(* Name: Nhat Ha Pham
   Student number: 547508*)

FUNCTION_BLOCK fbMaking_Coffee
VAR_INPUT
	GetOffBed : BOOL;  
	HeatButton : BOOL;
	Start : BOOL;
	ToastState : INT;
	Grinding : BOOL;
	Brewing : BOOL;
	Reset : BOOL;
	WaterError : BOOL;
END_VAR
VAR_OUTPUT
	WaterHotReady : BOOL;
	GrindingReady : BOOL;
	CoffeeWaitTime : BOOL;
	CoffeeMakingState : INT;
	CoffeeReady : BOOL;
	BrewingReady : BOOL;
	WaterLevelError : BOOL;
END_VAR
VAR
	WaterHot : BOOL;
	GrindingDone : BOOL;
	BrewingDone : BOOL;
	step: INT;
	TimerON : TON;   // Delay and creating wait time
	HeatingUp : BOOL;
	StartGrinding : BOOL;
	StartBrewing : BOOL;
END_VAR

(* Name: Nhat Ha Pham
   Student number: 547508*)

IF Reset THEN
	step := 0;
END_IF
CASE step OF
	0 : // Idle	
		WaterHotReady := FALSE;
		GrindingReady := FALSE;
		CoffeeWaitTime := FALSE;
		CoffeeReady := FALSE;
		BrewingReady := FALSE;
		CoffeeMakingState := 0;
		HeatButton := FALSE;
		Grinding := FALSE;
		Brewing := FALSE;
		WaterLevelError := FALSE;
		IF GetOffBed = TRUE AND Start THEN
			step := 10;
		END_IF
	10: // Start heating up the water
		IF HeatButton = TRUE THEN
			CoffeeMakingState := 1;
			HeatingUp := TRUE;
			CoffeeWaitTime := TRUE;   // Send a signal say need to wait 5s
		END_IF
		TimerON(IN := HeatingUp, PT := T#5S);   // Waiting the water being heated for 5s
		WaterHot := TimerON.Q;
		IF WaterHot THEN
			WaterHotReady := TRUE;
			HeatingUp := FALSE;
			CoffeeWaitTime := FALSE;   // Reset waiting signal
			step := 20;
			TimerON(IN := FALSE);   // Reset Timer
		END_IF
	20 : // Grind the coffee beans
		IF (ToastState = 1 OR ToastState = 2) AND Grinding THEN
			CoffeeMakingState := 2;
			CoffeeWaitTime := TRUE;   // Send a signal say need to wait 5s
			StartGrinding := TRUE;
		END_IF
		TimerON(IN := StartGrinding, PT := T#5S);
		GrindingDone := TimerON.Q;
		IF GrindingDone THEN
			GrindingReady := TRUE;
			StartGrinding := FALSE;
			CoffeeWaitTime := FALSE;   // Reset waiting signal
			step := 30;
			TimerON(IN := FALSE);   // // Reset Timer
		END_IF
	30 : //Brewing the coffee
		IF WaterError AND Brewing THEN
			step := 40;
		ELSIF ToastState = 2 AND Brewing AND NOT WaterError THEN
			StartBrewing := TRUE;
			CoffeeWaitTime := TRUE;
			CoffeeMakingState := 3;
		END_IF
		TimerON(IN := StartBrewing, PT := T#5S);
		BrewingDone := TimerON.Q;
		IF BrewingDone THEN
			BrewingReady := TRUE;
			StartBrewing := FALSE;
			CoffeeWaitTime := FALSE;   // Reset waiting signal
			CoffeeReady := TRUE;
			TimerON(IN := FALSE);   // // Reset Timer
		END_IF
		
	40 : // Error state
		WaterLevelError := TRUE;
END_CASE

END_FUNCTION_BLOCK

(* stored: Version 1.1.0.1, ProductVersion 3.1.4024.15
   POU fbMaking_Coffee: Id {6047ca55-2973-4800-b3c8-5ac6eb292b6c}, SpecialFunc None *)
